INTERFACE ITF_DigIn

METHOD get : BOOL
VAR_INPUT
END_VAR
END_METHOD

END_INTERFACE

(* stored: Version 1.1.0.1, ProductVersion 3.1.4026.8
   Itf ITF_DigIn: Id {ab9d6dbd-257f-46c0-83cf-c5d16120bcd5}
   Method get: Id {e5922c22-5820-401b-8741-c4a519e8766c} *)
